{attribute 'GeneratedUsingTerminal: AT2026-0250-0024'}
{attribute addProperty BoxType "AT2026-0250-0024"}
{attribute addProperty Id "A_0080_AT2002_5249_0019_AT2002_5249AT2002_33A3DF1B80"}
{attribute addProperty CRC "1908412773"}
{attribute addProperty Size "80"}
TYPE A_0068_AT2026_0250_0024_AT2026_0250_71C01165 EXTENDS AT2026_A7FEA1CF :
STRUCT
	{attribute addProperty Name "A_0080_AT2002_5249_0019_AT2002_5249"}
	{attribute addProperty PreviousPort "A_0068(AT2026-0250-0024) (AT2026-0250) : B"}
	A_0080_AT2002_5249_0019_AT2002_5249 : AT2002_33A3DF1B;
END_STRUCT
END_TYPE

(* stored: Version 1.2.0.0, ProductVersion 3.1.4024.9
   DUT A_0068_AT2026_0250_0024_AT2026_0250_71C01165: Id {feb92fa0-b4d4-4620-a20d-baed648099d2} *)
